// TIA Portal V20 export
// export: Created 2025-12-01T14:56:22.7552314Z, ExportSetting None, DisplayName Totally Integrated Automation Portal, DisplayVersion V20 Update 3, DisplayName TIA Portal Openness, DisplayVersion V20 Update 3, DisplayName TIA Portal Version Control Interface, DisplayVersion V20 Update 3, DisplayName STEP 7 Professional, DisplayVersion V20 Update 3, DisplayName STEP 7 Safety, DisplayVersion V20 Update 2, DisplayName WinCC Basic/Comfort/Advanced, DisplayVersion V20 Update 3, DisplayName WinCC Professional, DisplayVersion V20 Update 3, DisplayName WinCC Unified, DisplayVersion V20 Update 3
TYPE "ASI3_Diag_GW"
   STRUCT
      "Flags Fault Det" : Word;
      ConfigErrorsW0 : Word;
      ConfigErrorsW2 : Word;
      ConfigErrorsW4 : Word;
      ConfigErrorsW6 : Word;
      PeripheryFaultsW0 : Word;
      PeripheryFaultsW2 : Word;
      PeripheryFaultsW4 : Word;
      PeripheryFaultsW6 : Word;
   END_STRUCT;
END_TYPE
